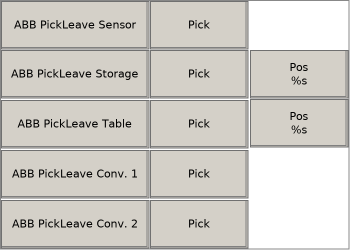
VISUALIZATION _VisuABBPickLeave  // 350x250
    Button (1,1 148x48), "ABB PickLeave Sensor"
        toggle ComGVL._fbTryOutABBPickLeaveSensorEn
    Button (1,50 148x48), "ABB PickLeave Storage"
        toggle ComGVL._fbTryOutABBPickLeaveStorageEn
    Button (1,100 148x48), "ABB PickLeave Table"
        toggle ComGVL._fbTryOutABBPickLeaveTableEn
    Button (1,150 148x48), "ABB PickLeave Conv. 1"
        toggle ComGVL._fbTryOutABBPickLeaveConveyor1En
    Button (1,200 148x48), "ABB PickLeave Conv. 2"
        toggle ComGVL._fbTryOutABBPickLeaveConveyor2En
    Button (150,1 98x48), "Pick"
        toggle ComGVL._fbTryOutABBPSensor
    Button (150,50 98x48), "Pick"
        toggle ComGVL._fbTryOutABBPStorage
    Button (150,100 98x48), "Pick"
        toggle ComGVL._fbTryOutABBPTable
    Button (150,150 98x48), "Pick"
        toggle ComGVL._fbTryOutABBPConveyor1
    Button (150,200 98x48), "Pick"
        toggle ComGVL._fbTryOutABBPConveyor2
    Button (250,50 98x48), "Pos %s", text variable: ComGVL._fbTryOutABBPStoragePos
        OnMouseClick: write the text variable via VisuDialogs.Numpad, min 1, max 9, title 'Position'
    Button (250,99 98x48), "Pos %s", text variable: ComGVL._fbTryOutABBPTablePos
        OnMouseClick: write the text variable via VisuDialogs.Numpad, min 1, max 9, title 'Position'
END_VISUALIZATION

(* stored: Version 1.1.0.1, ProductVersion 3.1.4024.2
   Visu _VisuABBPickLeave: Id {5806cf49-6c7d-47e3-995d-435f9acee2b5} *)
